// Mitsubishi GX Works2 project: Ex03   PLC: Q03UD

PROGRAM MAIN
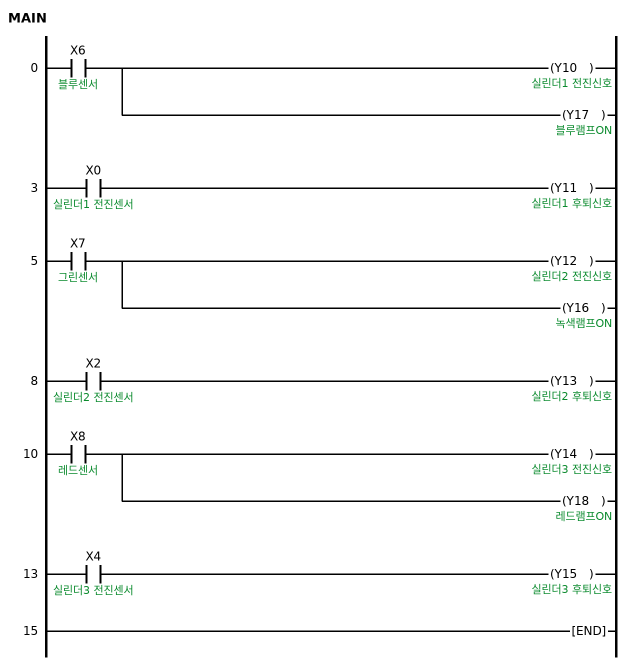
0     LD      X6  ; 블루센서
      OUT     Y10  ; 실린더1 전진신호
      OUT     Y17  ; 블루램프ON
3     LD      X0  ; 실린더1 전진센서
      OUT     Y11  ; 실린더1 후퇴신호
5     LD      X7  ; 그린센서
      OUT     Y12  ; 실린더2 전진신호
      OUT     Y16  ; 녹색램프ON
8     LD      X2  ; 실린더2 전진센서
      OUT     Y13  ; 실린더2 후퇴신호
10    LD      X8  ; 레드센서
      OUT     Y14  ; 실린더3 전진신호
      OUT     Y18  ; 레드램프ON
13    LD      X4  ; 실린더3 전진센서
      OUT     Y15  ; 실린더3 후퇴신호
15    END
END_PROGRAM

// device comments not shown above
X1  ; 실린더1 후진센서
X3  ; 실린더2 후진센서
X5  ; 실린더3 후진센서
